FUNCTION_BLOCK TURNTABLE_CTRL (* Basic Function Block Type *)
  (* Standard: 61499-2 *)
  (* Version 0.3, 2009-09-15, JHC, Holobloc Inc, Changed transition priorities. *)
  (* Version 0.2, 2003-12-04, JHC, Rockwell Automation, Renamed for better indexing. *)
  (* Version 0.1, 2002-11-05, JHC, Rockwell Automation, Corrected missing ST element in Algorithm REQ. *)
  (* Version 0.0, 2000-05-30, JHC, Rockwell Automation *)
  PACKAGE fb.rt.Conveyer;
  IMPORT fb.datatype.*;
  IMPORT fb.rt.*;
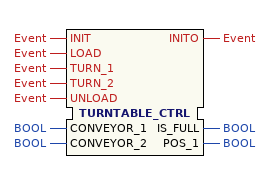
  EVENT_INPUT
    INIT; (* Initialization Request *)
    LOAD;
    TURN_1;
    TURN_2;
    UNLOAD;
  END_EVENT
  EVENT_OUTPUT
    INITO; (* Initialization Confirm *)
  END_EVENT
  VAR_INPUT
    CONVEYOR_1 : BOOL;
    CONVEYOR_2 : BOOL;
  END_VAR
  VAR_OUTPUT
    IS_FULL : BOOL;
    POS_1 : BOOL;
  END_VAR
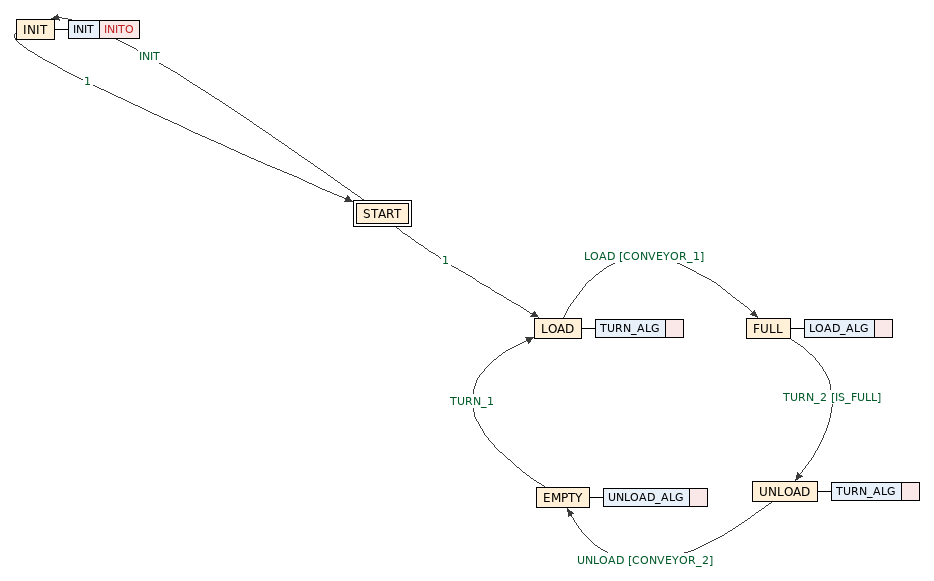
  EC_STATES
    START; (* Initial State *)
    INIT : INIT -> INITO; (* Initialization *)
    FULL : LOAD_ALG;
    LOAD : TURN_ALG;
    UNLOAD : TURN_ALG;
    EMPTY : UNLOAD_ALG;
  END_STATES
  EC_TRANSITIONS
    INIT TO START := 1;
    START TO INIT := INIT;
    START TO LOAD := 1;
    LOAD TO FULL := LOAD [CONVEYOR_1];
    UNLOAD TO EMPTY := UNLOAD [CONVEYOR_2];
    EMPTY TO LOAD := TURN_1;
    FULL TO UNLOAD := TURN_2 [IS_FULL];
  END_TRANSITIONS
  ALGORITHM INIT IN ST: (* Initialization algorithm *)
IS_FULL := FALSE;
POS_1 := FALSE;
CONVEYOR_1 := FALSE;
CONVEYOR_2 := FALSE;
  END_ALGORITHM
  ALGORITHM LOAD_ALG IN ST:
IS_FULL := TRUE;
  END_ALGORITHM
  ALGORITHM UNLOAD_ALG IN ST:
IS_FULL := FALSE;
  END_ALGORITHM
  ALGORITHM TURN_ALG IN ST:
IF POS_1 = TRUE THEN
	POS_1 := FALSE;
ELSE
	POS_1 := TRUE;
END_IF;
  END_ALGORITHM
END_FUNCTION_BLOCK
